FUNCTION_BLOCK makeAlarm
VAR
    alarm : REFERENCE TO p6com.AlarmDigital;
    onTime : TIME;
    offTime : TIME;

    onTimer : TON; 
    offTimer: TON;
    state : DINT;
 
END_VAR



onTimer(IN:= state=0, PT:= onTime);
offTimer(IN:= state=10, PT:= offTime);

CASE state OF
    0: 
        IF onTimer.Q THEN
            state := 10;
		END_IF
        
    10:
        IF offTimer.Q THEN
            state := 0;
		END_IF
END_CASE

alarm(ID:=2, IDName:='Alarm 1', Value := state = 10, TimeSpan := T#1MS);

METHOD FB_init : BOOL
VAR_INPUT
	bInitRetains : BOOL; // if TRUE, the retain variables are initialized (warm start / cold start)
	bInCopyCode : BOOL;  // if TRUE, the instance afterwards gets moved into the copy code (online change)
    alarm : REFERENCE TO p6com.AlarmDigital;
    onTime : TIME;
    offTime : TIME;
END_VAR
THIS^.alarm REF= alarm;
THIS^.onTime := onTime;
THIS^.offTime := offTime;
END_METHOD

END_FUNCTION_BLOCK

(* stored: Version 1.1.0.1, ProductVersion 3.1.4024.12
   POU makeAlarm: Id {68f2bc5a-2e92-4bd9-82e4-3d92820abdb6}, SpecialFunc None
   Method FB_init: Id {3a7c1f56-e97c-40ed-bc1f-bc5f0aba9381} *)
